// TIA Portal V16 export
// export: Created 2022-11-17T11:55:30.7316497Z, ExportSetting WithDefaults, DisplayName Totally Integrated Automation Portal, DisplayVersion V16 Update 6, DisplayName TIA Portal Version Control Interface, DisplayVersion V16 Update 2, DisplayName TIA Portal Openness, DisplayVersion V16 Update 6, DisplayName SINAMICS Startdrive Advanced, DisplayVersion V16 Update 5, DisplayName SINAMICS Startdrive G130, G150, S120, S150, SINAMICS MV, S210, DisplayVersion V16 Update 5, DisplayName SINAMICS Startdrive G110M, G120, G120C, G120D, G120P, G115D, DisplayVersion V16 Update 5, DisplayName STEP 7 Professional, DisplayVersion V16 Update 6, DisplayName STEP 7 Safety, DisplayVersion V16, DisplayName WinCC Advanced, DisplayVersion V16 Update 6
DATA_BLOCK "MB_REG1"   // DB201
{ S7_Optimized_Access := 'FALSE' }
VERSION : 0.1
// stored: AutoNumber false, IsOnlyStoredInLoadMemory false, IsWriteProtectedInAS false
   VAR RETAIN
      AD_R : UDInt := 40001;
      LN_R : UInt := 5;
      AD_W : UDInt := 0;
      LN_W : UInt := 0;
      A08R : Struct   // Prestiro_READ
         REG_0 : Int := 227;   // REG_CELLA
         REG_1 : Int := 24;   // REG_INPUT
         REG_2 : Int := 106;   // REG_VERSIONE
         REG_3 : Int := 0;   // REG_ENC1
         REG_4 : Int := 0;   // REG_ENC2
      END_STRUCT;
      A08W : Struct   // Prestiro_WRITE
         REG_5 : Int := 0;   // REG_OUTPUT1
         REG_6 : Int := 0;   // REG_OUTPUT2
         REG_7 : Int := 0;   // REG_OUTPUT3
         REG_8 : Int := 0;   // REG_ENCDIR
         REG_9 : Int := 0;
      END_STRUCT;
      SER : Struct   // Cordonatore_READ
         REG_10 : Int := 12337;
         REG_11 : Int := 12598;
         REG_12 : Int := 18480;
         REG_13 : Int := 12336;
         REG_14 : Int := 12592;
         REG_15 : Int := 0;
         REG_16 : Int := 0;
         REG_17 : Int := 0;
         REG_18 : Int := 0;
         REG_19 : Int := 0;
      END_STRUCT;
   END_VAR
BEGIN
END_DATA_BLOCK
